METHOD testValueIsNegative
VAR_INPUT
	(* for the test it's the parameter ``currentValue`` *)
	valueToTest	:LRealTestParameter;	
END_VAR
VAR
	(* just the expectation if the assertion to test must be worng or true *)
	assertionIsWrong		:BOOL;
	(* contains the format string for the test message *)
	message					:Tc2_System.T_MaxString;
	(* TwinCAT printf with the test message *)
	messageStringBuilder	:Tc2_Utilities.FB_FormatString;
	(* value of the paramter ``valueToTest`` as string *)
	valueToTestAsString		:Tc2_System.T_MaxString;
	(* binary value of the parameter ``valueToTest`` *)
	binaryValueToTest		:POINTER TO LWORD;
	(* sgin bit as BYTE for the message *)
	signBitAsByte			:BYTE;
	(* sgin bit as BOOL for the message *)
	signBit					:BOOL;	
END_VAR
THIS^.assertorContainer.resetAssertor();

binaryValueToTest := ADR(valueToTest.value);
signBit := binaryValueToTest^.SIGN;
signBitAsByte := TO_BYTE(signBit);
assertionIsWrong := (
	(NOT signBit)
	OR_ELSE Tc2_Utilities.LrealIsNaN(valueToTest.value)
);

message := SEL(
	assertionIsWrong,
	'currentValue is %s and sign bit is %u assertion must be TRUE', 
	'currentValue is %s and sign bit is %u assertion must be FALSE'
);

valueToTestAsString := valueToTest.asString;

messageStringBuilder(
	sFormat := message,
	arg1 := THIS^.AnyToArg(valueToTestAsString),
	arg2 := THIS^.AnyToArg(signBitAsByte)
);

THIS^.assertorContainer.assertor.assert.float.double.valueIsNegative(
	currentValue := valueToTest.value,
	message := ''
);

THIS^.AssertEquals_BOOL(
	Expected 	:= assertionIsWrong,
	Actual 		:= THIS^.assertorContainer.wasAssertionWrong,
	Message 	:= messageStringBuilder.sOut
);
END_METHOD

(*

short summary
==================
This test method tests ``assert.float.double.valueIsNegativeInfinite``
method of CNM_AssertionInterfaceLib library, 
it provides the possibility to handover test data via parameter 

.. <legal notes>

legal notes
=================
| SPDX-FileCopyrightText: © 2022 ekvip automation GmbH <info@ekvip.de>
| SPDX-License-Identifier: Apache-2.0
| For details check: Apache-2.0_

.. _Apache-2.0: https://www.apache.org/licenses/LICENSE-2.0

.. </legal notes>

parameters
==========

*)

METHOD testValueIsNegativeInfinite
VAR_INPUT
	(* for the test it's the parameter ``currentValue`` *)
	valueToTest	:LRealTestParameter;	
END_VAR
VAR
	(* just the expectation if the assertion to test must be worng or true *)
	assertionIsWrong		:BOOL;
	(* contains the format string for the test message *)
	message					:Tc2_System.T_MaxString;
	(* TwinCAT printf with the test message *)
	messageStringBuilder	:Tc2_Utilities.FB_FormatString;
	(* value of the paramter ``valueToTest`` as string *)
	valueToTestAsString		:Tc2_System.T_MaxString;
	(* binary value of the parameter ``valueToTest`` *)
	binaryValueToTest		:POINTER TO LWORD;
END_VAR
THIS^.assertorContainer.resetAssertor();

binaryValueToTest := ADR(valueToTest.value);
assertionIsWrong := (binaryValueToTest^ <> THIS^.BINARY_NEGATIVE_INFINITY);

message := SEL(
	assertionIsWrong,
	'currentValue is %s assertion must be TRUE', 
	'currentValue is %s assertion must be FALSE'
);

valueToTestAsString := valueToTest.asString;

messageStringBuilder(
	sFormat := message,
	arg1 := THIS^.AnyToArg(valueToTestAsString)
);

THIS^.assertorContainer.assertor.assert.float.double.valueIsNegativeInfinite(
	currentValue := valueToTest.value,
	message := ''
);

THIS^.AssertEquals_BOOL(
	Expected 	:= assertionIsWrong,
	Actual 		:= THIS^.assertorContainer.wasAssertionWrong,
	Message 	:= messageStringBuilder.sOut
);
END_METHOD

(*

short summary
==================
This test method tests ``assert.float.double.valueIsNegativeZero``
method of CNM_AssertionInterfaceLib library, 
it provides the possibility to handover test data via parameter 

.. <legal notes>

legal notes
=================
| SPDX-FileCopyrightText: © 2022 ekvip automation GmbH <info@ekvip.de>
| SPDX-License-Identifier: Apache-2.0
| For details check: Apache-2.0_

.. _Apache-2.0: https://www.apache.org/licenses/LICENSE-2.0

.. </legal notes>

parameters
==========

*)

METHOD testValueIsNegativeZero
VAR_INPUT
	(* for the test it's the parameter ``currentValue`` *)
	valueToTest	:LRealTestParameter;	
END_VAR
VAR
	(* just the expectation if the assertion to test must be worng or true *)
	assertionIsWrong		:BOOL;
	(* contains the format string for the test message *)
	message					:Tc2_System.T_MaxString;
	(* TwinCAT printf with the test message *)
	messageStringBuilder	:Tc2_Utilities.FB_FormatString;
	(* value of the paramter ``valueToTest`` as string *)
	valueToTestAsString		:Tc2_System.T_MaxString;
	(* binary value of the parameter ``valueToTest`` *)
	binaryValueToTest		:POINTER TO LWORD;
	(* sgin bit as BYTE for the message *)
	signBitAsByte			:BYTE;
	(* sgin bit as BOOL for the message *)
	signBit					:BOOL;	
END_VAR
THIS^.assertorContainer.resetAssertor();

binaryValueToTest := ADR(valueToTest.value);
signBit := binaryValueToTest^.SIGN;
signBitAsByte := TO_BYTE(signBit);

assertionIsWrong := (binaryValueToTest^ <> THIS^.BINARY_MINUS_ZERO);

message := SEL(
	assertionIsWrong,
	'currentValue is %s and sign bit is %u assertion must be TRUE', 
	'currentValue is %s and sign bit is %u assertion must be FALSE'
);

valueToTestAsString := valueToTest.asString;

messageStringBuilder(
	sFormat := message,
	arg1 := THIS^.AnyToArg(valueToTestAsString),
	arg2 := THIS^.AnyToArg(signBitAsByte)
);

THIS^.assertorContainer.assertor.assert.float.double.valueIsNegativeZero(
	currentValue := valueToTest.value,
	message := ''
);

THIS^.AssertEquals_BOOL(
	Expected 	:= assertionIsWrong,
	Actual 		:= THIS^.assertorContainer.wasAssertionWrong,
	Message 	:= messageStringBuilder.sOut
);
END_METHOD

(*

short summary
==================
This test method tests ``assert.float.double.valueIsNormal``
method of CNM_AssertionInterfaceLib library, 
it provides the possibility to handover test data via parameter 

.. <legal notes>

legal notes
=================
| SPDX-FileCopyrightText: © 2022 ekvip automation GmbH <info@ekvip.de>
| SPDX-License-Identifier: Apache-2.0
| For details check: Apache-2.0_

.. _Apache-2.0: https://www.apache.org/licenses/LICENSE-2.0

.. </legal notes>

parameters
==========

*)

METHOD testValueIsNormal
VAR_INPUT
	(* for the test it's the parameter ``currentValue`` *)
	valueToTest	:LRealTestParameter;	
END_VAR
VAR
	(* just the expectation if the assertion to test must be worng or true *)
	assertionIsWrong		:BOOL;
	(* contains the format string for the test message *)
	message					:Tc2_System.T_MaxString;
	(* TwinCAT printf with the test message *)
	messageStringBuilder	:Tc2_Utilities.FB_FormatString;
	(* value of the paramter ``valueToTest`` as string *)
	valueToTestAsString		:Tc2_System.T_MaxString;
	(* binary value of the parameter ``valueToTest`` *)
	binaryValueToTest		:POINTER TO LWORD;
END_VAR
THIS^.assertorContainer.resetAssertor();

binaryValueToTest := ADR(valueToTest.value);

assertionIsWrong := (
	((binaryValueToTest^ AND THIS^.MASK_FOR_EXPONENT) = THIS^.BINARY_ZERO)
	OR_ELSE Tc2_Utilities.LrealIsNaN(valueToTest.value)
	OR_ELSE (NOT Tc2_Utilities.LrealIsFinite(valueToTest.value))
);

message := SEL(
	assertionIsWrong,
	'currentValue is %s assertion must be TRUE', 
	'currentValue is %s assertion must be FALSE'
);

valueToTestAsString := valueToTest.asString;

messageStringBuilder(
	sFormat := message,
	arg1 := THIS^.AnyToArg(valueToTestAsString)
);

THIS^.assertorContainer.assertor.assert.float.double.valueIsNormal(
	currentValue := valueToTest.value,
	message := ''
);

THIS^.AssertEquals_BOOL(
	Expected 	:= assertionIsWrong,
	Actual 		:= THIS^.assertorContainer.wasAssertionWrong,
	Message 	:= messageStringBuilder.sOut
);
END_METHOD

(*

short summary
==================
This test method tests ``assert.float.double.valueIsNotEqualTo``
method of CNM_AssertionInterfaceLib library, 
it provides the possibility to handover test data via parameter 


.. <legal notes>

legal notes
=================
| SPDX-FileCopyrightText: © 2022 ekvip automation GmbH <info@ekvip.de>
| SPDX-License-Identifier: Apache-2.0
| For details check: Apache-2.0_

.. _Apache-2.0: https://www.apache.org/licenses/LICENSE-2.0

.. </legal notes>

parameters
==========

*)

METHOD testValueIsNotEqualTo 
VAR_INPUT
	(* for the test it's the parameter ``currentValue`` *)
	valueToTest		:LRealTestParameter;
	(* for the test it's the parameter ``unexpectedValue`` *)
	unexpectedValue	:LRealTestParameter;
	(* for the test it's the parameter ``tolerance`` *)
	tolerance		:LRealTestParameter;
END_VAR
VAR
	(* just the expectation if the assertion to test must be worng or true *)
	assertionIsWrong		:BOOL;
	(* contains the format string for the test message *)
	message					:Tc2_System.T_MaxString;
	(* TwinCAT printf with the test message *)
	messageStringBuilder	:Tc2_Utilities.FB_FormatString;
	(* just to cast *)
	binaryCurrentValue		:POINTER TO LWORD;
	(* just to cast *)
	binaryUnexpectedValue	:POINTER TO LWORD;
	(* value of the paramter ``valueToTest`` as string *)
	valueToTestAsString		:Tc2_System.T_MaxString;
	(* value of the paramter ``unexpectedValue`` as string *)
	unexpectedValueAsString	:Tc2_System.T_MaxString;
	(* value of the paramter ``tolerance`` as string *)
	toleranceAsString		:Tc2_System.T_MaxString;	
END_VAR
THIS^.assertorContainer.resetAssertor();
IF (
	Tc2_Utilities.LrealIsNaN(valueToTest.value)
	OR Tc2_Utilities.LrealIsNaN(unexpectedValue.value)
	OR Tc2_Utilities.LrealIsNaN(tolerance.value)
) THEN
	assertionIsWrong := FALSE;
ELSIF (NOT Tc2_Utilities.LrealIsFinite(tolerance.value)) THEN
	assertionIsWrong := TRUE;
ELSIF (
	Tc2_Utilities.LrealIsFinite(valueToTest.value)
	<> Tc2_Utilities.LrealIsFinite(unexpectedValue.value)
) THEN
	assertionIsWrong := FALSE; 
ELSIF (
	(NOT Tc2_Utilities.LrealIsFinite(valueToTest.value))
	OR (NOT Tc2_Utilities.LrealIsFinite(unexpectedValue.value))
) THEN
	binaryCurrentValue := ADR(valueToTest.value);
	binaryUnexpectedValue := ADR(unexpectedValue.value);
	assertionIsWrong := (binaryCurrentValue^.SIGN = binaryUnexpectedValue^.SIGN);
ELSE
	assertionIsWrong := (
		((unexpectedValue.value + ABS(tolerance.value)) >= valueToTest.value)
		AND ((unexpectedValue.value - ABS(tolerance.value)) <= valueToTest.value)
	);
END_IF

message := SEL(
	assertionIsWrong,
	'currentValue is %s unexpectedValue is %s tolerance is %s assertion must be TRUE', 
	'currentValue is %s unexpectedValue is %s tolerance is %s assertion must be FALSE'
);

valueToTestAsString := valueToTest.asString;
unexpectedValueAsString := unexpectedValue.asString;
toleranceAsString := tolerance.asString;

messageStringBuilder(
	sFormat := message,
	arg1 := THIS^.AnyToArg(valueToTestAsString),
	arg2 := THIS^.AnyToArg(unexpectedValueAsString),
	arg3 := THIS^.AnyToArg(toleranceAsString)
);

THIS^.assertorContainer.assertor.assert.float.double.valueIsNotEqualTo(
	currentValue	:= valueToTest.value,
	unexpectedValue	:= unexpectedValue.value,
	tolerance       := tolerance.value,
	message			:= ''
   );

THIS^.AssertEquals_BOOL(
	Expected 	:= assertionIsWrong,
	Actual 		:= THIS^.assertorContainer.wasAssertionWrong,
	Message 	:= messageStringBuilder.sOut
);
END_METHOD

(*

short summary
==================
This test method tests ``assert.float.double.valueIsNotNegativeInfinite``
method of CNM_AssertionInterfaceLib library, 
it provides the possibility to handover test data via parameter 

.. <legal notes>

legal notes
=================
| SPDX-FileCopyrightText: © 2022 ekvip automation GmbH <info@ekvip.de>
| SPDX-License-Identifier: Apache-2.0
| For details check: Apache-2.0_

.. _Apache-2.0: https://www.apache.org/licenses/LICENSE-2.0

.. </legal notes>

parameters
==========

*)

METHOD testValueIsNotNegativeInfinite
VAR_INPUT
	(* for the test it's the parameter ``currentValue`` *)
	valueToTest	:LRealTestParameter;	
END_VAR
VAR
	(* just the expectation if the assertion to test must be worng or true *)
	assertionIsWrong		:BOOL;
	(* contains the format string for the test message *)
	message					:Tc2_System.T_MaxString;
	(* TwinCAT printf with the test message *)
	messageStringBuilder	:Tc2_Utilities.FB_FormatString;
	(* value of the paramter ``valueToTest`` as string *)
	valueToTestAsString		:Tc2_System.T_MaxString;
	(* binary value of the parameter ``valueToTest`` *)
	binaryValueToTest		:POINTER TO LWORD;
END_VAR
THIS^.assertorContainer.resetAssertor();

binaryValueToTest := ADR(valueToTest.value);
assertionIsWrong := (binaryValueToTest^ = THIS^.BINARY_NEGATIVE_INFINITY);

message := SEL(
	assertionIsWrong,
	'currentValue is %s assertion must be TRUE', 
	'currentValue is %s assertion must be FALSE'
);

valueToTestAsString := valueToTest.asString;

messageStringBuilder(
	sFormat := message,
	arg1 := THIS^.AnyToArg(valueToTestAsString)
);

THIS^.assertorContainer.assertor.assert.float.double.valueIsNotNegativeInfinite(
	currentValue := valueToTest.value,
	message := ''
);

THIS^.AssertEquals_BOOL(
	Expected 	:= assertionIsWrong,
	Actual 		:= THIS^.assertorContainer.wasAssertionWrong,
	Message 	:= messageStringBuilder.sOut
);
END_METHOD

(*

short summary
==================
This test method tests ``assert.float.double.valueIsNotPositiveInfinite``
method of CNM_AssertionInterfaceLib library, 
it provides the possibility to handover test data via parameter 

.. <legal notes>

legal notes
=================
| SPDX-FileCopyrightText: © 2022 ekvip automation GmbH <info@ekvip.de>
| SPDX-License-Identifier: Apache-2.0
| For details check: Apache-2.0_

.. _Apache-2.0: https://www.apache.org/licenses/LICENSE-2.0

.. </legal notes>

parameters
==========

*)

METHOD testValueIsNotPositiveInfinite
VAR_INPUT
	(* for the test it's the parameter ``currentValue`` *)
	valueToTest	:LRealTestParameter;	
END_VAR
VAR
	(* just the expectation if the assertion to test must be worng or true *)
	assertionIsWrong		:BOOL;
	(* contains the format string for the test message *)
	message					:Tc2_System.T_MaxString;
	(* TwinCAT printf with the test message *)
	messageStringBuilder	:Tc2_Utilities.FB_FormatString;
	(* value of the paramter ``valueToTest`` as string *)
	valueToTestAsString		:Tc2_System.T_MaxString;
	(* binary value of the parameter ``valueToTest`` *)
	binaryValueToTest		:POINTER TO LWORD;
END_VAR
THIS^.assertorContainer.resetAssertor();

binaryValueToTest := ADR(valueToTest.value);
assertionIsWrong := (binaryValueToTest^ = THIS^.BINARY_INFINITY);

message := SEL(
	assertionIsWrong,
	'currentValue is %s assertion must be TRUE', 
	'currentValue is %s assertion must be FALSE'
);

valueToTestAsString := valueToTest.asString;

messageStringBuilder(
	sFormat := message,
	arg1 := THIS^.AnyToArg(valueToTestAsString)
);

THIS^.assertorContainer.assertor.assert.float.double.valueIsNotPositiveInfinite(
	currentValue := valueToTest.value,
	message := ''
);

THIS^.AssertEquals_BOOL(
	Expected 	:= assertionIsWrong,
	Actual 		:= THIS^.assertorContainer.wasAssertionWrong,
	Message 	:= messageStringBuilder.sOut
);
END_METHOD

(*

short summary
==================
This test method tests ``assert.float.double.valueIsNotSpecial``
method of CNM_AssertionInterfaceLib library, 
it provides the possibility to handover test data via parameter 

.. <legal notes>

legal notes
=================
| SPDX-FileCopyrightText: © 2022 ekvip automation GmbH <info@ekvip.de>
| SPDX-License-Identifier: Apache-2.0
| For details check: Apache-2.0_

.. _Apache-2.0: https://www.apache.org/licenses/LICENSE-2.0

.. </legal notes>

parameters
==========

*)

METHOD testValueIsNotSpecial
VAR_INPUT
	(* for the test it's the parameter ``currentValue`` *)
	valueToTest	:LRealTestParameter;	
END_VAR
VAR
	(* just the expectation if the assertion to test must be worng or true *)
	assertionIsWrong		:BOOL;
	(* contains the format string for the test message *)
	message					:Tc2_System.T_MaxString;
	(* TwinCAT printf with the test message *)
	messageStringBuilder	:Tc2_Utilities.FB_FormatString;
	(* value of the paramter ``valueToTest`` as string *)
	valueToTestAsString		:Tc2_System.T_MaxString;
END_VAR
THIS^.assertorContainer.resetAssertor();

assertionIsWrong := (
	(NOT Tc2_Utilities.LrealIsFinite(valueToTest.value))
	OR_ELSE Tc2_Utilities.LrealIsNaN(valueToTest.value)
);

message := SEL(
	assertionIsWrong,
	'currentValue is %s assertion must be TRUE', 
	'currentValue is %s assertion must be FALSE'
);

valueToTestAsString := valueToTest.asString;

messageStringBuilder(
	sFormat := message,
	arg1 := THIS^.AnyToArg(valueToTestAsString)
);

THIS^.assertorContainer.assertor.assert.float.double.valueIsNotSpecial(
	currentValue := valueToTest.value,
	message := ''
);

THIS^.AssertEquals_BOOL(
	Expected 	:= assertionIsWrong,
	Actual 		:= THIS^.assertorContainer.wasAssertionWrong,
	Message 	:= messageStringBuilder.sOut
);
END_METHOD

(*

short summary
==================
This test method tests ``assert.float.double.valueIsPositive``
method of CNM_AssertionInterfaceLib library, 
it provides the possibility to handover test data via parameter 

.. <legal notes>

legal notes
=================
| SPDX-FileCopyrightText: © 2022 ekvip automation GmbH <info@ekvip.de>
| SPDX-License-Identifier: Apache-2.0
| For details check: Apache-2.0_

.. _Apache-2.0: https://www.apache.org/licenses/LICENSE-2.0

.. </legal notes>

parameters
==========

*)

METHOD testValueIsPositive
VAR_INPUT
	(* for the test it's the parameter ``currentValue`` *)
	valueToTest	:LRealTestParameter;	
END_VAR
VAR
	(* just the expectation if the assertion to test must be worng or true *)
	assertionIsWrong		:BOOL;
	(* contains the format string for the test message *)
	message					:Tc2_System.T_MaxString;
	(* TwinCAT printf with the test message *)
	messageStringBuilder	:Tc2_Utilities.FB_FormatString;
	(* value of the paramter ``valueToTest`` as string *)
	valueToTestAsString		:Tc2_System.T_MaxString;
	(* binary value of the parameter ``valueToTest`` *)
	binaryValueToTest		:POINTER TO LWORD;
	(* sgin bit as BYTE for the message *)
	signBitAsByte			:BYTE;
	(* sgin bit as BOOL for the message *)
	signBit					:BOOL;	
END_VAR
THIS^.assertorContainer.resetAssertor();

binaryValueToTest := ADR(valueToTest.value);
signBit := binaryValueToTest^.SIGN;
signBitAsByte := TO_BYTE(signBit);
assertionIsWrong := (
	signBit
	OR Tc2_Utilities.LrealIsNaN(valueToTest.value)
);

message := SEL(
	assertionIsWrong,
	'currentValue is %s and sign bit is %u assertion must be TRUE', 
	'currentValue is %s and sign bit is %u assertion must be FALSE'
);

valueToTestAsString := valueToTest.asString;

messageStringBuilder(
	sFormat := message,
	arg1 := THIS^.AnyToArg(valueToTestAsString),
	arg2 := THIS^.AnyToArg(signBitAsByte)
);

THIS^.assertorContainer.assertor.assert.float.double.valueIsPositive(
	currentValue := valueToTest.value,
	message := ''
);

THIS^.AssertEquals_BOOL(
	Expected 	:= assertionIsWrong,
	Actual 		:= THIS^.assertorContainer.wasAssertionWrong,
	Message 	:= messageStringBuilder.sOut
);
END_METHOD

(*

short summary
==================
This test method tests ``assert.float.double.valueIsPositiveInfinite``
method of CNM_AssertionInterfaceLib library, 
it provides the possibility to handover test data via parameter 

.. <legal notes>

legal notes
=================
| SPDX-FileCopyrightText: © 2022 ekvip automation GmbH <info@ekvip.de>
| SPDX-License-Identifier: Apache-2.0
| For details check: Apache-2.0_

.. _Apache-2.0: https://www.apache.org/licenses/LICENSE-2.0

.. </legal notes>

parameters
==========

*)

METHOD testValueIsPositiveInfinite
VAR_INPUT
	(* for the test it's the parameter ``currentValue`` *)
	valueToTest	:LRealTestParameter;	
END_VAR
VAR
	(* just the expectation if the assertion to test must be worng or true *)
	assertionIsWrong		:BOOL;
	(* contains the format string for the test message *)
	message					:Tc2_System.T_MaxString;
	(* TwinCAT printf with the test message *)
	messageStringBuilder	:Tc2_Utilities.FB_FormatString;
	(* value of the paramter ``valueToTest`` as string *)
	valueToTestAsString		:Tc2_System.T_MaxString;
	(* binary value of the parameter ``valueToTest`` *)
	binaryValueToTest		:POINTER TO LWORD;
END_VAR
THIS^.assertorContainer.resetAssertor();

binaryValueToTest := ADR(valueToTest.value);
assertionIsWrong := (binaryValueToTest^ <> THIS^.BINARY_INFINITY);

message := SEL(
	assertionIsWrong,
	'currentValue is %s assertion must be TRUE', 
	'currentValue is %s assertion must be FALSE'
);

valueToTestAsString := valueToTest.asString;

messageStringBuilder(
	sFormat := message,
	arg1 := THIS^.AnyToArg(valueToTestAsString)
);

THIS^.assertorContainer.assertor.assert.float.double.valueIsPositiveInfinite(
	currentValue := valueToTest.value,
	message := ''
);

THIS^.AssertEquals_BOOL(
	Expected 	:= assertionIsWrong,
	Actual 		:= THIS^.assertorContainer.wasAssertionWrong,
	Message 	:= messageStringBuilder.sOut
);
END_METHOD

(*

short summary
==================
This test method tests ``assert.float.double.valueIsPositiveZero``
method of CNM_AssertionInterfaceLib library, 
it provides the possibility to handover test data via parameter 

.. <legal notes>

legal notes
=================
| SPDX-FileCopyrightText: © 2022 ekvip automation GmbH <info@ekvip.de>
| SPDX-License-Identifier: Apache-2.0
| For details check: Apache-2.0_

.. _Apache-2.0: https://www.apache.org/licenses/LICENSE-2.0

.. </legal notes>

parameters
==========

*)

METHOD testValueIsPositiveZero
VAR_INPUT
	(* for the test it's the parameter ``currentValue`` *)
	valueToTest	:LRealTestParameter;	
END_VAR
VAR
	(* just the expectation if the assertion to test must be worng or true *)
	assertionIsWrong		:BOOL;
	(* contains the format string for the test message *)
	message					:Tc2_System.T_MaxString;
	(* TwinCAT printf with the test message *)
	messageStringBuilder	:Tc2_Utilities.FB_FormatString;
	(* value of the paramter ``valueToTest`` as string *)
	valueToTestAsString		:Tc2_System.T_MaxString;
	(* binary value of the parameter ``valueToTest`` *)
	binaryValueToTest		:POINTER TO LWORD;
	(* sgin bit as BYTE for the message *)
	signBitAsByte			:BYTE;
	(* sgin bit as BOOL for the message *)
	signBit					:BOOL;	
END_VAR
THIS^.assertorContainer.resetAssertor();

binaryValueToTest := ADR(valueToTest.value);
signBit := binaryValueToTest^.SIGN;
signBitAsByte := TO_BYTE(signBit);

assertionIsWrong := (binaryValueToTest^ <> THIS^.BINARY_ZERO);

message := SEL(
	assertionIsWrong,
	'currentValue is %s and sign bit is %u assertion must be TRUE', 
	'currentValue is %s and sign bit is %u assertion must be FALSE'
);

valueToTestAsString := valueToTest.asString;

messageStringBuilder(
	sFormat := message,
	arg1 := THIS^.AnyToArg(valueToTestAsString),
	arg2 := THIS^.AnyToArg(signBitAsByte)
);

THIS^.assertorContainer.assertor.assert.float.double.valueIsPositiveZero(
	currentValue := valueToTest.value,
	message := ''
);

THIS^.AssertEquals_BOOL(
	Expected 	:= assertionIsWrong,
	Actual 		:= THIS^.assertorContainer.wasAssertionWrong,
	Message 	:= messageStringBuilder.sOut
);
END_METHOD

(*

short summary
==================
This test method tests ``assert.float.double.valueIsSpecial``
method of CNM_AssertionInterfaceLib library, 
it provides the possibility to handover test data via parameter 

.. <legal notes>

legal notes
=================
| SPDX-FileCopyrightText: © 2022 ekvip automation GmbH <info@ekvip.de>
| SPDX-License-Identifier: Apache-2.0
| For details check: Apache-2.0_

.. _Apache-2.0: https://www.apache.org/licenses/LICENSE-2.0

.. </legal notes>

parameters
==========

*)

METHOD testValueIsSpecial
VAR_INPUT
	(* for the test it's the parameter ``currentValue`` *)
	valueToTest	:LRealTestParameter;	
END_VAR
VAR
	(* just the expectation if the assertion to test must be worng or true *)
	assertionIsWrong		:BOOL;
	(* contains the format string for the test message *)
	message					:Tc2_System.T_MaxString;
	(* TwinCAT printf with the test message *)
	messageStringBuilder	:Tc2_Utilities.FB_FormatString;
	(* value of the paramter ``valueToTest`` as string *)
	valueToTestAsString		:Tc2_System.T_MaxString;
END_VAR
THIS^.assertorContainer.resetAssertor();

assertionIsWrong := (
	(NOT Tc2_Utilities.LrealIsNaN(valueToTest.value))
	AND_THEN (Tc2_Utilities.LrealIsFinite(valueToTest.value))
);

message := SEL(
	assertionIsWrong,
	'currentValue is %s assertion must be TRUE', 
	'currentValue is %s assertion must be FALSE'
);

valueToTestAsString := valueToTest.asString;

messageStringBuilder(
	sFormat := message,
	arg1 := THIS^.AnyToArg(valueToTestAsString)
);

THIS^.assertorContainer.assertor.assert.float.double.valueIsSpecial(
	currentValue := valueToTest.value,
	message := ''
);

THIS^.AssertEquals_BOOL(
	Expected 	:= assertionIsWrong,
	Actual 		:= THIS^.assertorContainer.wasAssertionWrong,
	Message 	:= messageStringBuilder.sOut
);
END_METHOD

(*

short summary
==================
This test method tests ``assert.float.double.valueIsSubnormal``
method of CNM_AssertionInterfaceLib library, 
it provides the possibility to handover test data via parameter 

.. <legal notes>

legal notes
=================
| SPDX-FileCopyrightText: © 2022 ekvip automation GmbH <info@ekvip.de>
| SPDX-License-Identifier: Apache-2.0
| For details check: Apache-2.0_

.. _Apache-2.0: https://www.apache.org/licenses/LICENSE-2.0

.. </legal notes>

parameters
==========

*)

METHOD testValueIsSubnormal
VAR_INPUT
	(* for the test it's the parameter ``currentValue`` *)
	valueToTest	:LRealTestParameter;	
END_VAR
VAR
	(* just the expectation if the assertion to test must be worng or true *)
	assertionIsWrong		:BOOL;
	(* contains the format string for the test message *)
	message					:Tc2_System.T_MaxString;
	(* TwinCAT printf with the test message *)
	messageStringBuilder	:Tc2_Utilities.FB_FormatString;
	(* value of the paramter ``valueToTest`` as string *)
	valueToTestAsString		:Tc2_System.T_MaxString;
	(* binary value of the parameter ``valueToTest`` *)
	binaryValueToTest		:POINTER TO LWORD;
END_VAR
THIS^.assertorContainer.resetAssertor();

binaryValueToTest := ADR(valueToTest.value);

assertionIsWrong := (
	((binaryValueToTest^ AND THIS^.MASK_FOR_EXPONENT) <> THIS^.BINARY_ZERO)
);

message := SEL(
	assertionIsWrong,
	'currentValue is %s assertion must be TRUE', 
	'currentValue is %s assertion must be FALSE'
);

valueToTestAsString := valueToTest.asString;

messageStringBuilder(
	sFormat := message,
	arg1 := THIS^.AnyToArg(valueToTestAsString)
);

THIS^.assertorContainer.assertor.assert.float.double.valueIsSubnormal(
	currentValue := valueToTest.value,
	message := ''
);

THIS^.AssertEquals_BOOL(
	Expected 	:= assertionIsWrong,
	Actual 		:= THIS^.assertorContainer.wasAssertionWrong,
	Message 	:= messageStringBuilder.sOut
);
END_METHOD

END_FUNCTION_BLOCK

(* stored: Version 1.1.0.1, ProductVersion 3.1.4024.12
   POU LRealAssertionTests: Id {4cdef9f6-aea7-47e1-a973-1a1e625cb7d9}, SpecialFunc None
   Folder internal: Id {55a78c18-c6f0-4b66-a6aa-792fa07f1e40}
   Folder valueIsANumber: Id {c9b81cb1-3d28-4c93-b044-b859fef34f8d}
   Folder valueIsEqualTo: Id {cb34475c-b4d7-42a5-bd9e-15c700b2806e}
   Folder valueIsFinite: Id {5c0c9d31-6210-40f2-b1ab-4667167ca000}
   Folder valueIsGreaterThan: Id {ffa6b16a-871b-43ef-8dde-4d6eee078ea1}
   Folder valueIsInfinite: Id {863226ec-1e47-4545-b043-cfa078beab65}
   Folder valueIsInRangeOf: Id {237c4a1b-299e-432c-9b8c-3ea021088efc}
   Folder valueIsLessThan: Id {462e0175-fd69-4d14-ab10-4cb34cefd812}
   Folder valueIsMax: Id {b3a473d0-e1aa-4a22-8661-42298afa5290}
   Folder valueIsMin: Id {3d02cbf4-1326-4c23-baf3-a2eea53014b5}
   Folder valueIsNaN: Id {c71a9c78-4843-49c1-bce1-9bd76d1a646b}
   Folder valueIsNegative: Id {3dcb3e65-0417-4c17-bf15-eb8504e9c8d3}
   Folder valueIsNegativeZero: Id {fce9c057-8072-4a48-b835-1f3394ec4c1e}
   Folder valueIsNegInfinite: Id {8f95f117-a915-4daa-808c-be94399d9b0e}
   Folder valueIsNormal: Id {48943a1c-d523-4c2f-8247-1f0b6d57eea3}
   Folder valueIsNotEqualTo: Id {b4bacf5d-61b3-46f5-8320-06568e53cc2b}
   Folder valueIsNotNegInf: Id {00012e42-5d5f-4a60-bc55-131907fb72a6}
   Folder valueIsNotPosInf: Id {7ff6c67b-baa7-4f0e-a513-c43cef34b606}
   Folder valueIsNotSpecial: Id {bf8d6ef0-edeb-4e1a-86ee-3747b12ee906}
   Folder valueIsPosInfinite: Id {30b69d2b-d974-4d67-a6e2-29b2a04b3540}
   Folder valueIsPositive: Id {a00449ba-37d2-4545-b648-be16d4e64c4d}
   Folder valueIsPositiveZero: Id {bc6b203b-48cd-4459-bdda-9f03812395d1}
   Folder valueIsSpecial: Id {cb32aef4-2d4d-4812-8b85-3f75ff4178cd}
   Folder valueIsSubnormal: Id {266fbcbc-518f-417c-ad7a-817d5f144ea7}
   Method FB_init: Id {39816376-de75-40d7-b4de-febbec9bb1e7}
   Method getTestNameFor: Id {618c4f00-1437-4fdc-a957-5e323f3ae1cc}
   Method runValueIsANumberTests: Id {32293ef8-5339-4531-a969-4cef8cd4acfd}
   Method runValueIsEqualToTests: Id {de4bad80-9c96-4fff-a086-3e74441d3c1d}
   Method runValueIsFiniteTests: Id {ef83ab90-0dcf-4724-8ea5-80da6724b357}
   Method runValueIsGreaterThanTests: Id {c69faa20-08c5-46d4-8c1f-b1ab3cdadb74}
   Method runValueIsInfiniteTests: Id {589e72b1-fe49-429e-8df6-b1a6a046c863}
   Method runValueIsInRangeOfTests: Id {3ed90c21-5f02-473b-98a5-03b8857c1550}
   Method runValueIsLessThanTests: Id {bbe8b0f1-0d80-43ce-9a39-18b5cc1f207b}
   Method runValueIsMaxTests: Id {b1c919c7-15ce-414f-a451-53d585cdfbea}
   Method runValueIsMinTests: Id {56aa7749-9f36-422b-956a-3faef2c5a138}
   Method runValueIsNaNTests: Id {75129fd3-8cfb-4d75-87c8-a0bba0cd63c5}
   Method runValueIsNegativeInfiniteTests: Id {67ef3164-f1f6-4671-94d8-25d1ff634672}
   Method runValueIsNegativeTests: Id {97a5f293-8c8e-4183-8cc5-f86158b211ce}
   Method runValueIsNegativeZeroTests: Id {b4fb472c-f608-443d-b454-10a003aca9b2}
   Method runValueIsNormalTests: Id {b609c3ae-6540-49dd-8d90-e4ffdb81c765}
   Method runValueIsNotEqualToTests: Id {f02af843-ea77-4244-96fa-5e99ad5eeb88}
   Method runValueIsNotNegativeInfiniteTests: Id {385586b3-3ffa-4192-8684-25dfa2c22d7b}
   Method runValueIsNotPositiveInfiniteTests: Id {d67b6e20-bfb0-4c4a-8032-6a6af7af56f7}
   Method runValueIsNotSpecialTests: Id {4d61ebf3-1386-4c40-80c6-d67d50a5d56d}
   Method runValueIsPositiveInfiniteTests: Id {5a24b56a-5648-4901-a8b8-cd3d17bc5f78}
   Method runValueIsPositiveTests: Id {c0e52967-a5ef-485f-9dc5-54a0bb67890c}
   Method runValueIsPositiveZeroTests: Id {06928a47-9f2a-42a8-a787-c67cd059b79a}
   Method runValueIsSpecialTests: Id {67b3e52f-f7e4-448b-bb74-7cbff11c2d13}
   Method runValueIsSubnormalTests: Id {8cb68382-0bcf-4a85-bbaa-50952f0f0fd1}
   Method testValueIsANumber: Id {40956583-6a76-41fa-810f-1175f18c7652}
   Method testValueIsEqualTo: Id {74336c2f-8fb6-418a-8d9d-eb99470ec2e7}
   Method testValueIsFinite: Id {56a3c1e8-9430-404c-b828-bf3eb2626b22}
   Method testValueIsGreaterThan: Id {3ee2ce96-cf79-45a6-ae11-2149cd0051cc}
   Method testValueIsInfinite: Id {6d4a316c-5e31-4431-9786-d65e34723f6b}
   Method testValueIsInRangeOf: Id {964ffdf5-0066-45ac-94ac-3c32080a745a}
   Method testValueIsLessThan: Id {14d72b7e-616f-400b-95be-5ad6407bcabd}
   Method testValueIsMax: Id {5a6939c4-e05b-499e-958c-954e3529a3fb}
   Method testValueIsMin: Id {8c96d293-0120-4ff0-9bcf-86cf16be9877}
   Method testValueIsNaN: Id {6b9908e3-c23c-4144-9d37-a6dacd09c856}
   Method testValueIsNegative: Id {24e2b382-be5d-4d91-99ff-557e4eb71055}
   Method testValueIsNegativeInfinite: Id {afdadbc7-259f-471b-9f5f-99eeaf9ab7cd}
   Method testValueIsNegativeZero: Id {8b073e02-d2c5-4878-bb11-5e1013a4a8d9}
   Method testValueIsNormal: Id {721ff8f1-1a16-4813-a33d-c2a62a217f5f}
   Method testValueIsNotEqualTo: Id {2a425286-606d-42e7-8621-5c05450cb403}
   Method testValueIsNotNegativeInfinite: Id {335f2f08-5d81-4eb7-932b-c5e5234ad541}
   Method testValueIsNotPositiveInfinite: Id {d4a60b2f-0668-4746-9882-2daf4ccd02d6}
   Method testValueIsNotSpecial: Id {cc64d524-f1c3-413f-81b6-011c3699970a}
   Method testValueIsPositive: Id {c46e15a1-6558-4fc3-b9f6-aceb4e148962}
   Method testValueIsPositiveInfinite: Id {bac3cf27-4dd6-4d01-9d6a-fd77b35bb536}
   Method testValueIsPositiveZero: Id {63313205-3682-4c15-bbf7-178b1b16ffb8}
   Method testValueIsSpecial: Id {76b71d9d-6664-4a93-a2ae-bd05c9f1d61a}
   Method testValueIsSubnormal: Id {b778b55e-1817-44e0-8edb-30fb2d3923be} *)
